FUNCTION_BLOCK ASSEMBLE_AQ_FROM_AX (* assembles 2 AX (BOOL) adapters into one 2-bit AQ adapter *)
  (* Standard: 61499-2; Description: Copyright (c) 2026 Meisterschulen am Ostbahnhof SPDX-License-Identifier: EPL-2.0 *)
  (* Version 1.0, 2026-05-16, Franz Höpfinger, Meisterschulen am Ostbahnhof, Initial Version *)
  PACKAGE adapter::assembling;
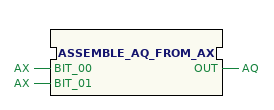
  SOCKETS
    BIT_00 : adapter::types::unidirectional::AX; (* Bit 0 *)
    BIT_01 : adapter::types::unidirectional::AX; (* Bit 1 *)
  END_SOCKETS
  PLUGS
    OUT : adapter::types::unidirectional::AQ; (* AQ Output *)
  END_PLUGS
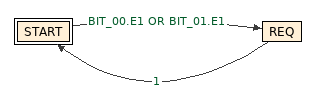
  EC_STATES
    START;
    REQ;
  END_STATES
  EC_TRANSITIONS
    START TO REQ := BIT_00.E1 OR BIT_01.E1;
    REQ TO START := 1;
  END_TRANSITIONS
  ALGORITHM REQ IN ST:
OUT.D1 := BYTE#0;
OUT.D1.%X0 := BIT_00.D1;
OUT.D1.%X1 := BIT_01.D1;
OUT.E1();
  END_ALGORITHM
END_FUNCTION_BLOCK
(* other elements stored in the file *)
(* Algorithm Name=REQ *)
